// TIA Portal V16 export
// export: Created 2024-09-05T17:39:24.3071184Z, ExportSetting WithDefaults, DisplayName Totally Integrated Automation Portal, DisplayVersion V16 Update 6, DisplayName TIA Portal Version Control Interface, DisplayVersion V16 Update 2, DisplayName TIA Portal Openness, DisplayVersion V16 Update 6, DisplayName STEP 7 Professional, DisplayVersion V16 Update 6, DisplayName STEP 7 Safety, DisplayVersion V16, DisplayName WinCC Advanced, DisplayVersion V16 Update 6
FUNCTION_BLOCK "6. Call_M004_NTRS"   // FB2006, LAD
{ S7_Optimized_Access := 'TRUE' }
AUTHOR : bartz
VERSION : 0.1
// stored: AutoNumber false, IsIECCheckEnabled false, IsRetainMemResEnabled false, MemoryReserve 100, SetENOAutomatically false, UDAEnableTagReadback false
   VAR_INPUT
      nTRSTag : Bool;
      TIMESTAMP_IN { ExternalAccessible := 'False'; ExternalVisible := 'False'; ExternalWritable := 'False'} : WString;
   END_VAR
   VAR
      nTRSTagTemp : Bool;
   END_VAR
BEGIN

REGION Network 1 (SCL)
   IF #nTRSTag <> #nTRSTagTemp THEN

       "MII_Interface_Data".MII_METHODS.M004_NTRS.Inputs.PLC_ID := "MII_Parameters".Connection.PLC_ID;
       "MII_Interface_Data".MII_METHODS.M004_NTRS.Inputs.PLANT := "MII_Parameters".Connection.PlantID;
       "MII_Interface_Data".MII_METHODS.M004_NTRS.Inputs.STOPPAGE := #nTRSTag;

       // New from version 4a
       "MII_Interface_Data".MII_METHODS.M004_NTRS.Inputs.TIMESTAMP := #TIMESTAMP_IN;

       //Call the method 
       "1. DMC_setConnection_DB".CallBuffer[6] := TRUE;

       #nTRSTagTemp := #nTRSTag;
   END_IF;
END_REGION
END_FUNCTION_BLOCK
